Universal Robots URScript: command03.urscript

def leanForwardJoint():
  movej([0.4537856055,-2.00712864,-2.059488517,-0.6457718232,1.570796327,2.024581932], a=5.0, v=1.0)
end
